# EPICS substitutions: elioApp/Db/EL3154.substitutions
file EL3154.template { pattern
{ CHAN	}
{ 1	}
{ 2	}
{ 3	}
{ 4	}
}
